# EPICS IOC start-up script: iocsh/ethercatmc2slit_hard.iocsh
dbLoadRecords("ethercatmcslit_hard.template", "P=$(P), SLIT=$(SLIT), mXp=$(mXp), mXn=$(mXn), mXc=$(mXc), mXg=$(mXg) ")
